(* PLC project Unnamed, Unknown Unnamed 1 *)
(* stored: creationDateTime 2026-05-06T15:04:10, modificationDateTime 2026-05-06T15:04:10 *)

PROGRAM main
  VAR
    PushBtn AT %IX0.0 : BOOL;
    LEDBlue AT %QX0.0 : BOOL;
    LEDGreen AT %QX0.1 : BOOL;
    LEDYellow AT %QX0.2 : BOOL;
    LEDRed AT %QX0.3 : BOOL;
  END_VAR
  VAR
    DebounceTime : TIME := T#50ms;
    ledNo : INT;
    BtnDelay : BOOL;
    TONBtnDelay : TON;
    BtnTrigger : R_TRIG;
    triggerReset : BOOL;
    CountUpLEDNo : CTU;
    LEDRed_Active : BOOL := FALSE;
    LEDYellow_Active : BOOL := FALSE;
    LEDGreen_Active : BOOL;
    LEDBlue_Active : BOOL;
    R_TRIG0 : R_TRIG;
    pulseReset : BOOL;
  END_VAR
  VAR  (* added by the conversion: wires and edge detectors of the diagram *)
    _GT531915_OUT : BOOL;
    _GT531915_ENO : BOOL;
  END_VAR

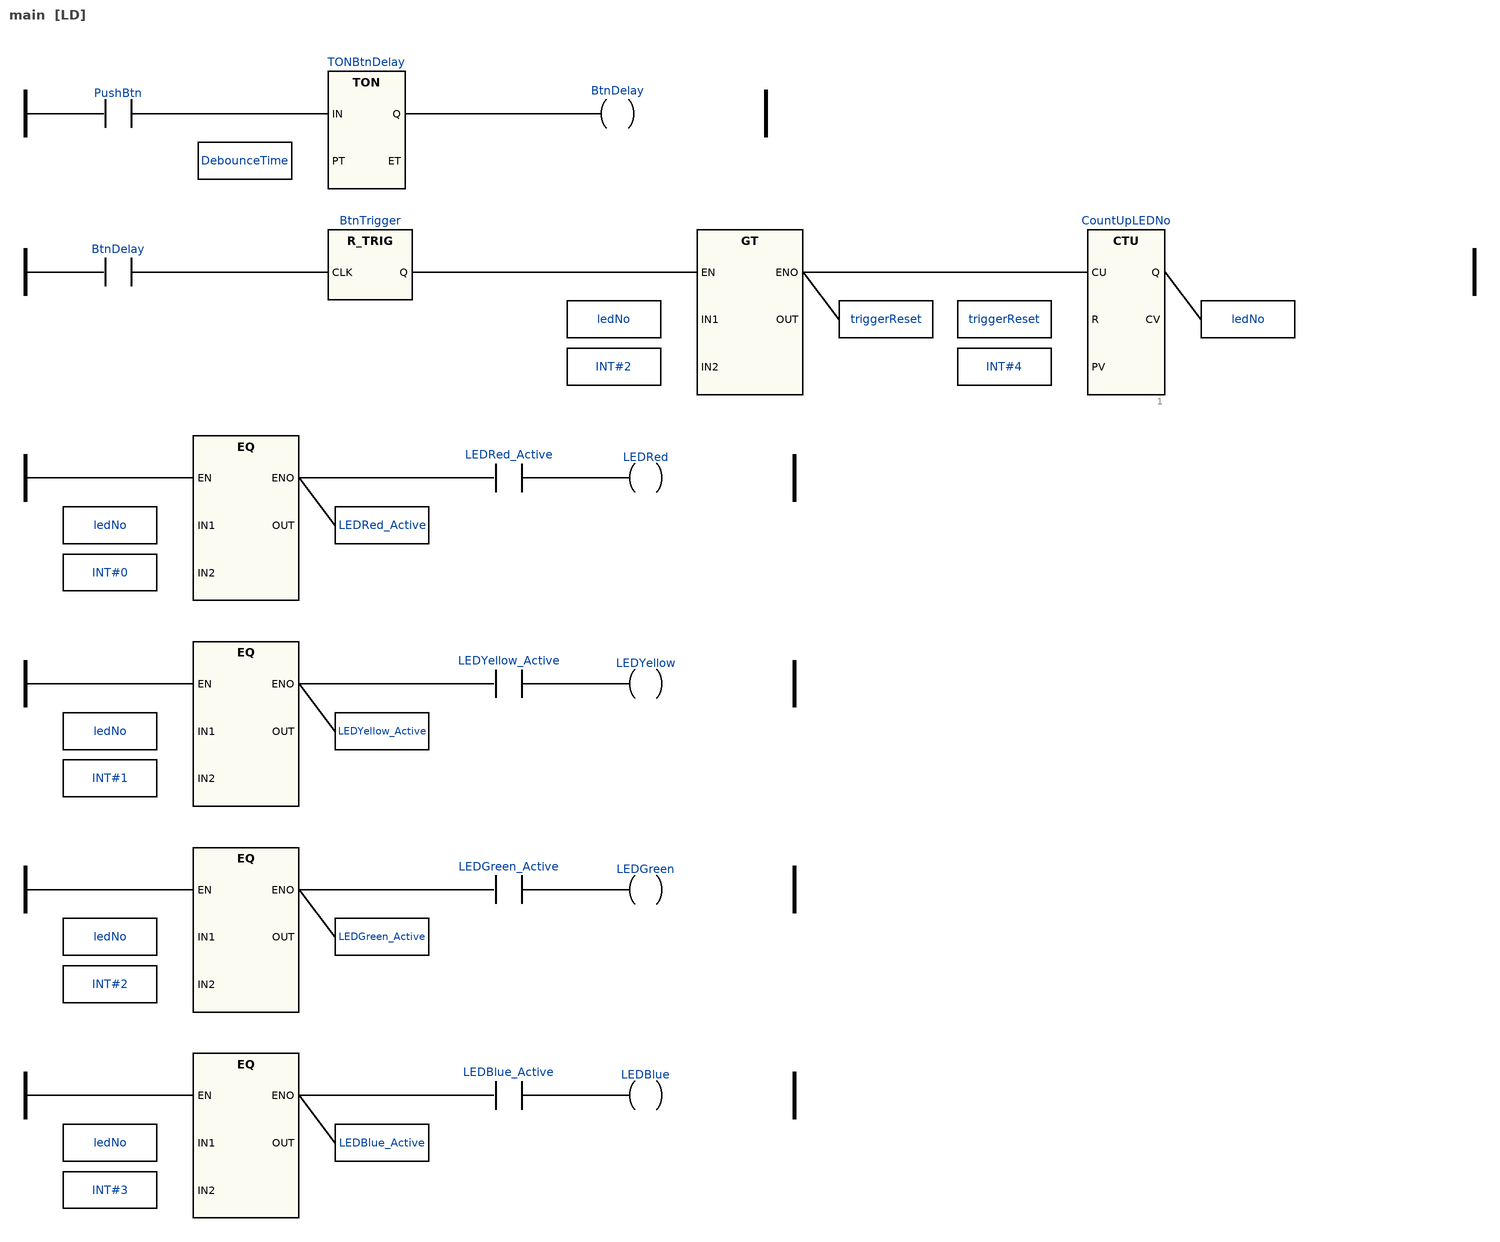
(* LD diagram, written out as Structured Text *)
CountUpLEDNo(CU := _GT531915_OUT, R := triggerReset, PV := INT#4);
TONBtnDelay(IN := PushBtn, PT := DebounceTime);
BtnDelay := TONBtnDelay.Q;
LEDRed := LEDRed_Active;
LEDYellow := LEDYellow_Active;
LEDGreen := LEDGreen_Active;
LEDBlue := LEDBlue_Active;
BtnTrigger(CLK := BtnDelay);
_GT531915_OUT := GT(EN := BtnTrigger.Q, IN1 := ledNo, IN2 := INT#2, ENO => _GT531915_ENO);
IF _GT531915_ENO THEN triggerReset := _GT531915_OUT; END_IF;
ledNo := CountUpLEDNo.CV;
LEDRed_Active := ledNo = INT#0;
LEDYellow_Active := ledNo = INT#1;
LEDGreen_Active := ledNo = INT#2;
LEDBlue_Active := ledNo = INT#3;
END_PROGRAM

CONFIGURATION Config0
  RESOURCE Res0 ON PLC
    TASK task0(INTERVAL := T#20ms, PRIORITY := 1);
    PROGRAM instance0 WITH task0 : main;
  END_RESOURCE
END_CONFIGURATION
